% RSLogix 500 project CLOCK_BAK034.RSS, saved by version 8.30.00.16 %
PROJECT "UNTITLED"    % processor: MicroLogix 1000 %

PROGRAM FILES
  LAD 2 "MAIN_PROG"  12 rungs
  LAD 3 "USER_FAULT"  1 rungs
  LAD 4 "HSC_INT"  1 rungs
  LAD 5 "STI_INT"  1 rungs
  LAD 6, 7, 8, 9, 10, 11, 12, 13, 14, 15, 16: only END

DATA FILES
  O0 OUTPUT  1 elements
  I1 INPUT  2 elements
  S2 STATUS  33 elements
  B3 BINARY  32 elements
  T4 TIMER  40 elements
  C5 COUNTER  32 elements
  R6 CONTROL  16 elements
  N7 INTEGER  105 elements

LADDER 2 "MAIN_PROG"
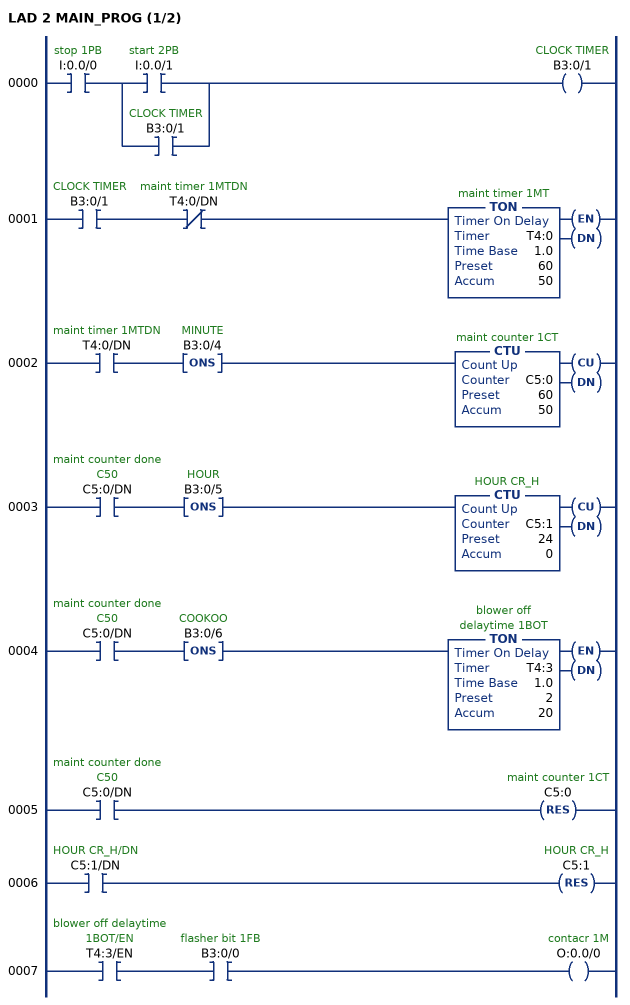
% Rung: 0 %
SOR XIC I:0.0/0 BST XIC I:0.0/1 NXB XIC B3:0/1 BND OTE B3:0/1 EOR
%   I:0.0/0  1PB  "stop" %
%   I:0.0/1  2PB  "start" %
%   B3:0/1  "CLOCK TIMER" %
% Rung: 1 %
SOR XIC B3:0/1 XIO T4:0/DN TON T4:0 1.0 60 50 EOR
%   B3:0/1  "CLOCK TIMER" %
%   T4:0/DN  1MTDN  "maint timer" %
%   T4:0  1MT  "maint timer" %
% Rung: 2 %
SOR XIC T4:0/DN OSR B3:0/4 CTU C5:0 60 50 EOR
%   T4:0/DN  1MTDN  "maint timer" %
%   B3:0/4  "MINUTE" %
%   C5:0  1CT  "maint counter" %
% Rung: 3 %
SOR XIC C5:0/DN OSR B3:0/5 CTU C5:1 24 0 EOR
%   C5:0/DN  C50  "maint counter done" %
%   B3:0/5  "HOUR" %
%   C5:1  CR_H  "HOUR" %
% Rung: 4 %
SOR XIC C5:0/DN OSR B3:0/6 TON T4:3 1.0 2 20 EOR
%   C5:0/DN  C50  "maint counter done" %
%   B3:0/6  "COOKOO" %
%   T4:3  1BOT  "blower off delaytime" %
% Rung: 5 %
SOR XIC C5:0/DN RES C5:0 EOR
%   C5:0/DN  C50  "maint counter done" %
%   C5:0  1CT  "maint counter" %
% Rung: 6 %
SOR XIC C5:1/DN RES C5:1 EOR
%   C5:1  CR_H  "HOUR" %
% Rung: 7 %
SOR XIC T4:3/EN XIC B3:0/0 OTE O:0.0/0 EOR
%   T4:3  1BOT  "blower off delaytime" %
%   B3:0/0  1FB  "flasher bit" %
%   O:0.0/0  1M  "contacr" %

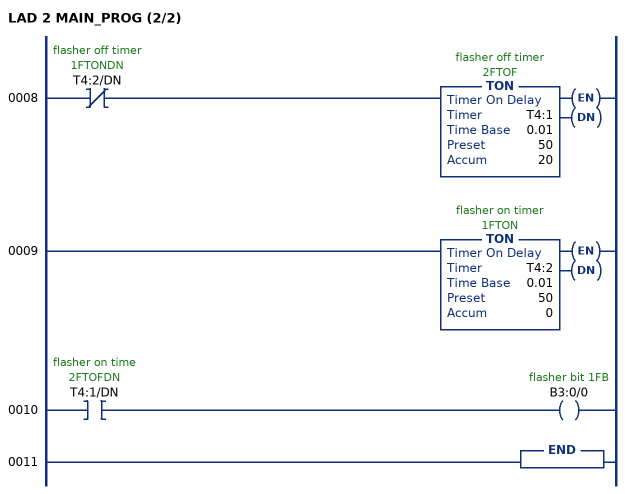
% Rung: 8 %
SOR XIO T4:2/DN TON T4:1 0.01 50 20 EOR
%   T4:2/DN  1FTONDN  "flasher off timer" %
%   T4:1  2FTOF  "flasher off timer" %
% Rung: 9 %
SOR TON T4:2 0.01 50 0 EOR
%   T4:2  1FTON  "flasher on timer" %
% Rung: 10 %
SOR XIC T4:1/DN OTE B3:0/0 EOR
%   T4:1/DN  2FTOFDN  "flasher on time" %
%   B3:0/0  1FB  "flasher bit" %
% Rung: 11 %
SOR END EOR

OTHER DOCUMENTED ADDRESSES
  B3:4  "MINUTE OSR"
  B3:5  "HOUR OSR"
  B3:6  "COOKOO"
  I:0.0/2  PB  "maint timer rest"
  I:0.0/3  3PB  "maint timer rest"
  I:0.0/4  4PB  "maint counter reset"
  O:0.0/1  1LT  "motor off"
  O:0.0/2  2LT  "motor on"
  O:0.0/3  3LT  "maint light"
  O:0.0/4  1BM  "blower motor"
  T4  
  T4:3/DN  "blower off delay timer"

DATA TABLE (non-zero values as saved)
DATA T4
% .PRE .ACC %
% T4:0 % 60 50
% T4:1 % 50 20
% T4:2 % 50 0
% T4:3 % 2 20
DATA C5
% .PRE .ACC %
% C5:0 % 60 50
% C5:1 % 24 0
